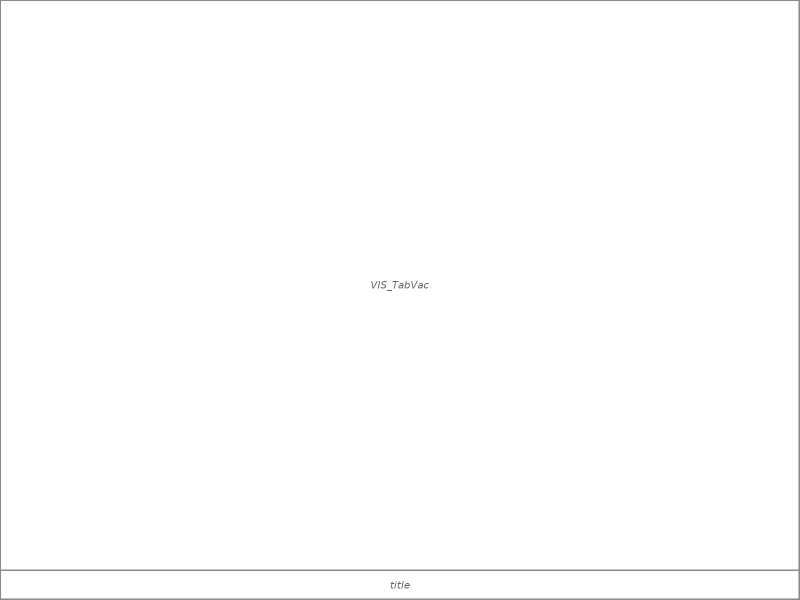
VISUALIZATION F3_MediaTransport  // 800x600
    TabControl (0,0 800x570)
        shows VIS_TabVac()
        shows VIS_UpDownSlot()
        [0]: TabTitle=TabVac
        [1]: TabTitle=UpDownSlot
    Frame (0,570 800x30)
        shows title()
END_VISUALIZATION

(* stored: Version 1.1.0.1, ProductVersion 3.1.4024.11
   Visu F3_MediaTransport: Id {dfd9df58-16a7-4787-ac45-1fec26d8c029} *)
